(****************************************************************************************)
(*							Beckhoff Automation Poland									*)
(*								FB_TypeSR  v1											*)
(*									27.05.2008											*)
(*				Bloczek przerzutnika SR	(przewaga SET)									*)
(*______________________________________________________________________________________*)
FUNCTION_BLOCK FB_TypeSR
VAR_INPUT
	bR:			BOOL;
	bS:			BOOL;
END_VAR
VAR_OUTPUT
	bQ:			BOOL;
END_VAR
VAR
END_VAR

IF(bS=1) THEN bQ:=1;
ELSIF(bR=1) THEN bQ:=0;
END_IF

END_FUNCTION_BLOCK

(* stored: Version 1.1.0.1, ProductVersion 3.1.4020.3
   POU FB_TypeSR: Id {164dabca-5c6e-4c45-8813-834ae2986628}, SpecialFunc None *)
